FUNCTION_BLOCK FB_EtherCATCheck
VAR_INPUT
END_VAR
VAR_OUTPUT
END_VAR
VAR
	//drive EtherCAT communition detection
	m_commuEtherCATState:FB_EcGetSlaveState;
	m_EcSlaveState : ST_EcSlaveState;
	
	m_crcVerify : FB_EcGetSlaveCrcError;
	m_crcError : ST_EcCrcError;
	
	m_EtherCATVerify : ST_EtherCATState;
END_VAR

METHOD EtherCATVerify : ST_EtherCATState
VAR_INPUT
	armsNetID:T_AmsNetID;
	jntAddr:UINT;
END_VAR

m_commuEtherCATState(sNetId:= armsNetID, nSlaveAddr:= jntAddr, bExecute:= TRUE, tTimeout:= , bBusy=> , bError=> , nErrId=> , state=> m_EcSlaveState);

IF NOT m_commuEtherCATState.bBusy THEN
	m_commuEtherCATState(bExecute:=FALSE);
	IF m_EcSlaveState.deviceState = EC_DEVICE_STATE_OP THEN
		m_EtherCATVerify.EtherCATState := TRUE;
	ELSE
		m_EtherCATVerify.EtherCATState := FALSE;
	END_IF
END_IF


m_crcVerify(sNetId:= armsNetID, nSlaveAddr:= jntAddr, bExecute:= TRUE, tTimeout:= , bBusy=> , bError=> , nErrId=> , crcError=> m_crcError);
IF NOT m_crcVerify.bBusy THEN
	m_crcVerify(bExecute:=FALSE);
	m_EtherCATVerify.CRCPortA := MAX(EtherCATVerify.CRCPortA,m_crcError.portA);
	m_EtherCATVerify.CRCPortB := MAX(EtherCATVerify.CRCPortB,m_crcError.portB);
	m_EtherCATVerify.CRCPortC := MAX(EtherCATVerify.CRCPortC,m_crcError.portC);
END_IF

EtherCATVerify := m_EtherCATVerify;
END_METHOD

END_FUNCTION_BLOCK

(* stored: Version 1.1.0.1, ProductVersion 3.1.4024.11
   POU FB_EtherCATCheck: Id {439b82da-b334-4605-8920-d50ed36120b2}, SpecialFunc None
   Method EtherCATVerify: Id {700221e4-3451-4ebe-a364-9420b7ed5cfc} *)
